// TIA Portal V19 export
DATA_BLOCK "TCON_DI"   // DB365
// stored: AutoNumber false, InstanceOfName TCON, OfSystemLibElement TCON, OfSystemLibVersion 4.0
"TCON"
   // VAR_INPUT
   //    REQ : Bool := TRUE;
   //    ID : CONN_OUC := 16#0002;
   // END_VAR
   // VAR_OUTPUT
   //    DONE : Bool := TRUE;
   //    BUSY : Bool := FALSE;
   //    ERROR : Bool := FALSE;
   //    STATUS : Word := 16#0000;
   // END_VAR
   // VAR_IN_OUT
   //    CONNECT : Variant;
   // END_VAR
BEGIN
END_DATA_BLOCK
